PROGRAM PRG_CommandHandler
VAR
    // ================================================================
    // 1. COMMAND & STATE FLAGS
    // ================================================================
    bisValidCmd           : BOOL;
    bCancelCmd            : BOOL;
    bHome                 : BOOL;
    bisLinearActuator     : BOOL;
    bisLinearTableHomeCmd : BOOL;
    bisLinearTableMoveCmd : BOOL;
    bisResetCmd           : BOOL;

    bOperationInProgress  : BOOL := FALSE;
    bCancelInProgress     : BOOL := FALSE;
    CancelMove            : BOOL := FALSE;
    bSafetyOk             : BOOL := FALSE;
    bAwaitingHMIClose     : BOOL := FALSE;

    // ================================================================
    // 2. REFERENCES TO FUNCTION BLOCKS / STRUCTURES
    // ================================================================
    LinearActuator    : POINTER TO FB_LinearActuator;
    LinearTable       : POINTER TO FB_StepperMotor;
    LinearActuatorCmd : POINTER TO ST_LinearActuatorCommand;
    LinearTableCmd    : POINTER TO ST_StepperMotorCommand;

    // ================================================================
    // 3. INPUTS / PARAMETERS
    // ================================================================
    nX                 : SINT;
    sY                 : STRING;
    sZ                 : STRING;
    sRequestedActuator : STRING := '';

    // ================================================================
    // 4. OUTPUTS / RESULTS
    // ================================================================
    CurrentPosition : LREAL;
    Result          : INT := 0;
    nCancelResult   : INT := 0;

    // ================================================================
    // 5. LOOP / TEMP VARIABLES
    // ================================================================
    i : INT;

    // ================================================================
    // 6. TIMERS
    // ================================================================
    tmrCancelTimeout   : TON;
    tCancelTimeout     : TIME := T#5S;

    tmrHMICloseSignal  : TON;
    tHMICloseHoldTime  : TIME := T#1000MS;
END_VAR

(* 1. SAFETY CHECK *)
bSafetyOk := EvaluateSystemSafety();

(* 2. WAIT FOR HMI TO EXIT COMMAND PROMPT *)
IF bAwaitingHMIClose THEN
	// Start timer
    tmrHMICloseSignal(IN := TRUE, PT := tHMICloseHoldTime);
    
	// Timer expired
    IF tmrHMICloseSignal.Q THEN     
        sRequestedActuator := 'none';
        bAwaitingHMIClose := FALSE;
        tmrHMICloseSignal(IN := FALSE);
    END_IF
    
    RETURN;
END_IF

(* 3. COMMAND CANCEL LOGIC *)
IF CancelMove AND bOperationInProgress AND NOT bCancelInProgress THEN
    bCancelInProgress := TRUE;
END_IF

IF bCancelInProgress THEN
    ProcessCancelOperation();
	
    RETURN; 
END_IF

(* 4. PROCESS NEW COMMAND *)
bisValidCmd := F_ValidateCommand(sInput := sRequestedActuator, nX => nX, sY => sY, sZ => sZ);

IF NOT bOperationInProgress AND sRequestedActuator <> 'none' AND sRequestedActuator <> 'close' AND (bSafetyOk OR IsResetCommand(sZ)) THEN
  
    IF NOT bisValidCmd THEN      
        sRequestedActuator := 'close';
        bAwaitingHMIClose := TRUE;
        tmrHMICloseSignal(IN := FALSE); 
		
        RETURN; 
    END_IF
    
	bOperationInProgress := TRUE;
    
	// Get command data
    LinearActuator := F_GetLinearCommandValue(nX, sY);
    LinearActuatorCmd := F_GetLinearCommandMember(nX, sY);
    LinearTable := F_GetStepperCommandValue(nX, sY);
    LinearTableCmd := F_GetStepperCommandMember(nX, sY);
    
	// Set command type
    bisLinearActuator := sY = 'Chariot' OR sY = 'Compressor' OR sY = 'Sensor' OR sY = 'HeatExCoupola' OR sY = 'RegenCoupola';  
    bisLinearTableHomeCmd := sY = 'Home' AND LinearTableCmd^.Homing;
    bisLinearTableMoveCmd := sY = 'Motor';
    bisResetCmd := sZ = 'Reset';
END_IF

(* 5. EXECUTE COMMAND *)
IF bOperationInProgress AND NOT bCancelInProgress THEN
	
    IF bisLinearActuator THEN
        ProcessLinearActuator();
    ELSIF bisLinearTableHomeCmd THEN
        ProcessLinearTable(bHome := TRUE);
    ELSIF bisLinearTableMoveCmd THEN
        ProcessLinearTable(bHome := FALSE);
    END_IF
	
END_IF

METHOD EvaluateSystemSafety : BOOL
EvaluateSystemSafety := TRUE;

FOR i := 1 TO 5 DO
    EvaluateSystemSafety := EvaluateSystemSafety AND gSystemAlarmStatus.aZoneStatus[i].bOkToRun;
END_FOR
END_METHOD

METHOD IsResetCommand : BOOL
VAR_INPUT
    sResetFlag : STRING;  
END_VAR
IF sResetFlag = 'Reset' THEN
    IsResetCommand := TRUE;
ELSE
	// Default behavior
    IsResetCommand := bSafetyOk;
END_IF
END_METHOD


METHOD ProcessCancelOperation
VAR
    bCancelComplete : BOOL := FALSE;
    bTimeoutExpired : BOOL := FALSE;
    bSafetyTimeoutExpired : BOOL := FALSE;
END_VAR
IF bisLinearActuator THEN
    nCancelResult := LinearActuator^.Cancel();
	
    CASE nCancelResult OF
        1: // Success
			LinearActuatorCmd^.Status := -2;
			
       -1: // Failure
			LinearActuatorCmd^.Status := -1;
    END_CASE;

    bCancelComplete := (nCancelResult <> 0);

ELSIF bisLinearTableHomeCmd OR bisLinearTableMoveCmd THEN
    nCancelResult := LinearTable^.Stop(TRUE);

    CASE nCancelResult OF
        1: // Success
            LinearTable^.GetPosition(fCurrentPosition => CurrentPosition);
            LinearTableCmd^.Position := CurrentPosition;
            
            IF bisLinearTableHomeCmd THEN
                LinearTableCmd^.Homed := FALSE;
                LinearTableCmd^.Homing := FALSE;
            END_IF;

            bCancelComplete := TRUE;

       -1: // Failure
            IF bisLinearTableHomeCmd THEN
                LinearTableCmd^.Homed := FALSE;
                LinearTableCmd^.Homing := FALSE;
            ELSE
                LinearTableCmd^.Position := -1;
            END_IF;

            bCancelComplete := TRUE;
    END_CASE;
END_IF;

// Cleanup
IF bCancelComplete THEN
	sRequestedActuator := 'close';
	bAwaitingHMIClose := TRUE;
	tmrHMICloseSignal(IN := FALSE); 

    bOperationInProgress := FALSE;
    bCancelInProgress := FALSE;
    CancelMove := FALSE;
    nCancelResult := 0;
END_IF
END_METHOD

METHOD ProcessLinearActuator
VAR
	bisExtendCmd : BOOL;
END_VAR
// Get command value
bisExtendCmd := LinearActuatorCmd^.Command;

(* 1. RESET COMMAND CHECK *)
IF bisResetCmd THEN
    LinearActuator^.Reset(State => Result); // Instantaneous read of prox seonsors
	
    bOperationInProgress := FALSE;
	
	sRequestedActuator := 'close';
    bAwaitingHMIClose := TRUE;
    tmrHMICloseSignal(IN := FALSE); 
	
    RETURN;
END_IF

(* 2. EXECUTE MOVEMENT COMMAND *)
IF bisExtendCmd THEN
    Result := LinearActuator^.Extend();
ELSE
    Result := LinearActuator^.Home();
END_IF

CASE Result OF
    1: // Success
        bOperationInProgress := FALSE;
        
        IF bisExtendCmd THEN
            LinearActuatorCmd^.Status := 1;
        ELSE
            LinearActuatorCmd^.Status := 0;
        END_IF
        
        sRequestedActuator := 'close';
        bAwaitingHMIClose := TRUE;
        tmrHMICloseSignal(IN := FALSE); 
    
    0: // Continue
        // Operation in progress
        
   -1: // Failure
        bOperationInProgress := FALSE;
		
        LinearActuatorCmd^.Status := -1;
        
        sRequestedActuator := 'close';
        bAwaitingHMIClose := TRUE;
        tmrHMICloseSignal(IN := FALSE); 
END_CASE
END_METHOD

METHOD ProcessLinearTable
VAR_INPUT
	bHome : BOOL;
END_VAR
// Get command value
LinearTable^.GetPosition(fCurrentPosition => CurrentPosition);

(* 1. RESET COMMAND CHECK *)
IF bisResetCmd THEN
    Result := LinearTable^.Reset(TRUE);
    
    CASE Result OF
        1: // Success

            bOperationInProgress := FALSE;
			
            LinearTableCmd^.Position := CurrentPosition;
            
            sRequestedActuator := 'close';
            bAwaitingHMIClose := TRUE;
            tmrHMICloseSignal(IN := FALSE); 
			
            RETURN;
            
        0: // Continue
            // Operation in progress
            
       -1: // Failure
            bOperationInProgress := FALSE;
			
            LinearTableCmd^.Position := -1;
            
            sRequestedActuator := 'close';
            bAwaitingHMIClose := TRUE;
            tmrHMICloseSignal(IN := FALSE);
			
            RETURN;
    END_CASE
END_IF

(* 2. EXECUTE MOVEMENT COMMAND *)
IF bHome THEN
    Result := LinearTable^.Home(TRUE);
ELSE
    Result := LinearTable^.MoveToPosition(fPosition := LinearTableCmd^.Command);
    LinearTableCmd^.Position := CurrentPosition;
END_IF

CASE Result OF
    1: // Success
        bOperationInProgress := FALSE;
        
        IF bHome THEN    
            LinearTableCmd^.Homed := TRUE;
            LinearTableCmd^.Homing := FALSE;
        END_IF
        
        sRequestedActuator := 'close';
        bAwaitingHMIClose := TRUE;
        tmrHMICloseSignal(IN := FALSE);
    		
    0: // Continue
        // Operation in progress
    
   -1: // Failure
        bOperationInProgress := FALSE;
        
        IF bHome THEN    
            LinearTableCmd^.Homed := FALSE;
            LinearTableCmd^.Homing := FALSE;
        ELSE
            LinearTableCmd^.Position := -1;
        END_IF
        
        sRequestedActuator := 'close';
        bAwaitingHMIClose := TRUE;
        tmrHMICloseSignal(IN := FALSE); 
END_CASE
END_METHOD

END_PROGRAM

(* stored: Version 1.1.0.1, ProductVersion 3.1.4026.11
   POU PRG_CommandHandler: Id {b534ce1c-328a-4a1f-bd2e-b4f58fd46cee}, SpecialFunc None
   Method EvaluateSystemSafety: Id {9dd680db-6fdd-4722-ae01-3267e2a2aa12}
   Method IsResetCommand: Id {b06412f3-9a53-431c-82a1-ed0a29a747c2}
   Method ProcessCancelOperation: Id {ac957e77-13a6-4f5c-8c3f-8b6fbdb8d91f}
   Method ProcessLinearActuator: Id {fa11d454-59c0-4fad-b564-0953d0ce78c6}
   Method ProcessLinearTable: Id {b89bcaac-8269-4091-97df-2a76137525f9} *)
